REGION Network 172: M875- / M23-SWITCH ON SPINDLE FRAME BLOWING
   RUNG wire#powerrail
      Contact( "DB339_EXTENDED_M_SPARE".M_code[875] )
      wire#w1
      I_Contact( "DB371_M_UNIT_SPARE".M_CODES_SPARE.Ack_M875 )
      I_Contact( "DB2120_MPP_ITC_IPC".RESET_FAULTS )
      I_Contact( "DB371_M_UNIT_SPARE".M_CODES_SPARE.M_RESET_PULSE )
      Coil( "DB371_M_UNIT_SPARE".M_CODES_SPARE.M875 )
   END_RUNG
   RUNG wire#powerrail
      Contact( "DB371_M_UNIT_SPARE".M_CODES_SPARE.M875 )
   END_RUNG wire#w1
   // the same network as SCL:
   "DB371_M_UNIT_SPARE".M_CODES_SPARE.M875 := ("DB339_EXTENDED_M_SPARE".M_code[875] OR "DB371_M_UNIT_SPARE".M_CODES_SPARE.M875) AND NOT "DB371_M_UNIT_SPARE".M_CODES_SPARE.Ack_M875 AND NOT "DB2120_MPP_ITC_IPC".RESET_FAULTS AND NOT "DB371_M_UNIT_SPARE".M_CODES_SPARE.M_RESET_PULSE;
END_REGION

REGION Network 173: ACKNOWLEDGE M888- / ACKNOWLEDGE M23-SWITCH ON SPINDLE FRAME BLOWING
   RUNG wire#powerrail
      Contact( "M_ZERO" )
      Coil( "DB371_M_UNIT_SPARE".M_CODES_SPARE.Ack_M888 )
   END_RUNG
   // the same network as SCL:
   "DB371_M_UNIT_SPARE".M_CODES_SPARE.Ack_M888 := "M_ZERO";
END_REGION

REGION Network 174: M888- / M23-SWITCH ON SPINDLE FRAME BLOWING
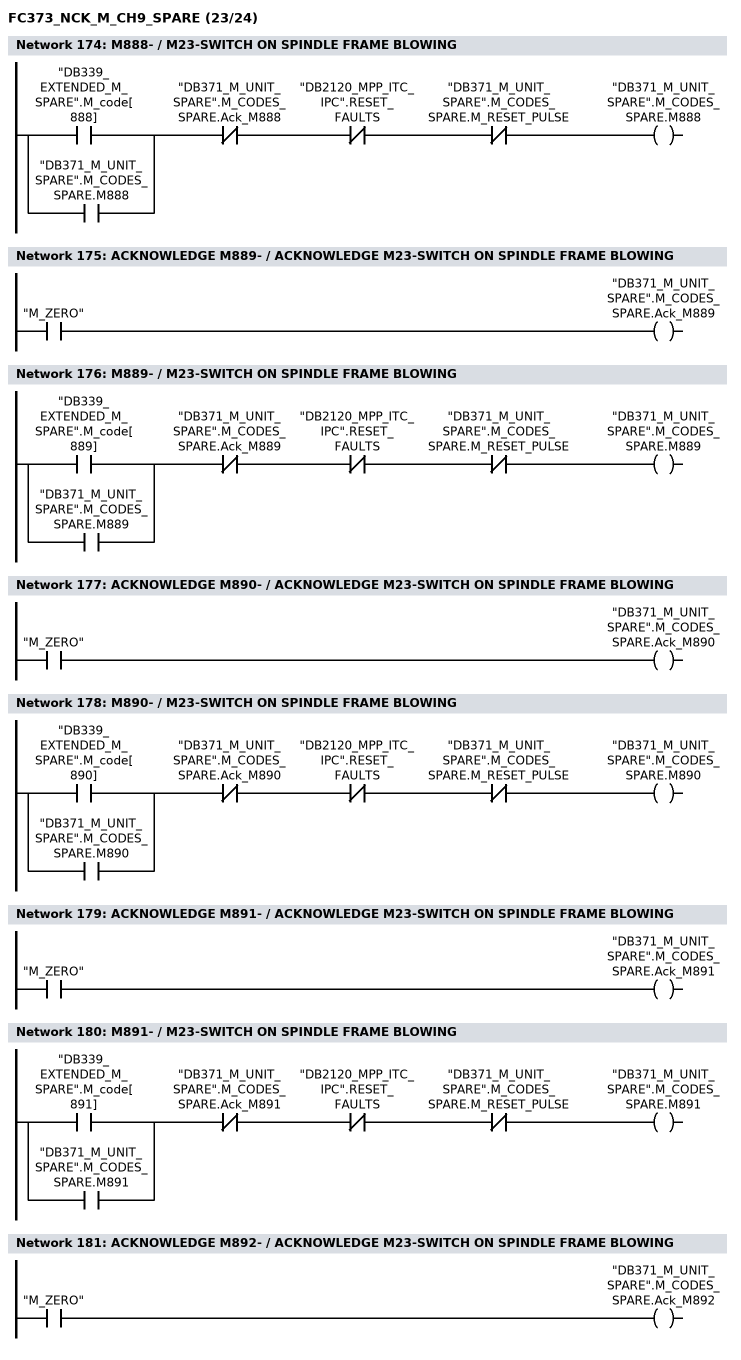
   RUNG wire#powerrail
      Contact( "DB339_EXTENDED_M_SPARE".M_code[888] )
      wire#w1
      I_Contact( "DB371_M_UNIT_SPARE".M_CODES_SPARE.Ack_M888 )
      I_Contact( "DB2120_MPP_ITC_IPC".RESET_FAULTS )
      I_Contact( "DB371_M_UNIT_SPARE".M_CODES_SPARE.M_RESET_PULSE )
      Coil( "DB371_M_UNIT_SPARE".M_CODES_SPARE.M888 )
   END_RUNG
   RUNG wire#powerrail
      Contact( "DB371_M_UNIT_SPARE".M_CODES_SPARE.M888 )
   END_RUNG wire#w1
   // the same network as SCL:
   "DB371_M_UNIT_SPARE".M_CODES_SPARE.M888 := ("DB339_EXTENDED_M_SPARE".M_code[888] OR "DB371_M_UNIT_SPARE".M_CODES_SPARE.M888) AND NOT "DB371_M_UNIT_SPARE".M_CODES_SPARE.Ack_M888 AND NOT "DB2120_MPP_ITC_IPC".RESET_FAULTS AND NOT "DB371_M_UNIT_SPARE".M_CODES_SPARE.M_RESET_PULSE;
END_REGION

REGION Network 175: ACKNOWLEDGE M889- / ACKNOWLEDGE M23-SWITCH ON SPINDLE FRAME BLOWING
   RUNG wire#powerrail
      Contact( "M_ZERO" )
      Coil( "DB371_M_UNIT_SPARE".M_CODES_SPARE.Ack_M889 )
   END_RUNG
   // the same network as SCL:
   "DB371_M_UNIT_SPARE".M_CODES_SPARE.Ack_M889 := "M_ZERO";
END_REGION

REGION Network 176: M889- / M23-SWITCH ON SPINDLE FRAME BLOWING
   RUNG wire#powerrail
      Contact( "DB339_EXTENDED_M_SPARE".M_code[889] )
      wire#w1
      I_Contact( "DB371_M_UNIT_SPARE".M_CODES_SPARE.Ack_M889 )
      I_Contact( "DB2120_MPP_ITC_IPC".RESET_FAULTS )
      I_Contact( "DB371_M_UNIT_SPARE".M_CODES_SPARE.M_RESET_PULSE )
      Coil( "DB371_M_UNIT_SPARE".M_CODES_SPARE.M889 )
   END_RUNG
   RUNG wire#powerrail
      Contact( "DB371_M_UNIT_SPARE".M_CODES_SPARE.M889 )
   END_RUNG wire#w1
   // the same network as SCL:
   "DB371_M_UNIT_SPARE".M_CODES_SPARE.M889 := ("DB339_EXTENDED_M_SPARE".M_code[889] OR "DB371_M_UNIT_SPARE".M_CODES_SPARE.M889) AND NOT "DB371_M_UNIT_SPARE".M_CODES_SPARE.Ack_M889 AND NOT "DB2120_MPP_ITC_IPC".RESET_FAULTS AND NOT "DB371_M_UNIT_SPARE".M_CODES_SPARE.M_RESET_PULSE;
END_REGION

REGION Network 177: ACKNOWLEDGE M890- / ACKNOWLEDGE M23-SWITCH ON SPINDLE FRAME BLOWING
   RUNG wire#powerrail
      Contact( "M_ZERO" )
      Coil( "DB371_M_UNIT_SPARE".M_CODES_SPARE.Ack_M890 )
   END_RUNG
   // the same network as SCL:
   "DB371_M_UNIT_SPARE".M_CODES_SPARE.Ack_M890 := "M_ZERO";
END_REGION

REGION Network 178: M890- / M23-SWITCH ON SPINDLE FRAME BLOWING
   RUNG wire#powerrail
      Contact( "DB339_EXTENDED_M_SPARE".M_code[890] )
      wire#w1
      I_Contact( "DB371_M_UNIT_SPARE".M_CODES_SPARE.Ack_M890 )
      I_Contact( "DB2120_MPP_ITC_IPC".RESET_FAULTS )
      I_Contact( "DB371_M_UNIT_SPARE".M_CODES_SPARE.M_RESET_PULSE )
      Coil( "DB371_M_UNIT_SPARE".M_CODES_SPARE.M890 )
   END_RUNG
   RUNG wire#powerrail
      Contact( "DB371_M_UNIT_SPARE".M_CODES_SPARE.M890 )
   END_RUNG wire#w1
   // the same network as SCL:
   "DB371_M_UNIT_SPARE".M_CODES_SPARE.M890 := ("DB339_EXTENDED_M_SPARE".M_code[890] OR "DB371_M_UNIT_SPARE".M_CODES_SPARE.M890) AND NOT "DB371_M_UNIT_SPARE".M_CODES_SPARE.Ack_M890 AND NOT "DB2120_MPP_ITC_IPC".RESET_FAULTS AND NOT "DB371_M_UNIT_SPARE".M_CODES_SPARE.M_RESET_PULSE;
END_REGION

REGION Network 179: ACKNOWLEDGE M891- / ACKNOWLEDGE M23-SWITCH ON SPINDLE FRAME BLOWING
   RUNG wire#powerrail
      Contact( "M_ZERO" )
      Coil( "DB371_M_UNIT_SPARE".M_CODES_SPARE.Ack_M891 )
   END_RUNG
   // the same network as SCL:
   "DB371_M_UNIT_SPARE".M_CODES_SPARE.Ack_M891 := "M_ZERO";
END_REGION

REGION Network 180: M891- / M23-SWITCH ON SPINDLE FRAME BLOWING
   RUNG wire#powerrail
      Contact( "DB339_EXTENDED_M_SPARE".M_code[891] )
      wire#w1
      I_Contact( "DB371_M_UNIT_SPARE".M_CODES_SPARE.Ack_M891 )
      I_Contact( "DB2120_MPP_ITC_IPC".RESET_FAULTS )
      I_Contact( "DB371_M_UNIT_SPARE".M_CODES_SPARE.M_RESET_PULSE )
      Coil( "DB371_M_UNIT_SPARE".M_CODES_SPARE.M891 )
   END_RUNG
   RUNG wire#powerrail
      Contact( "DB371_M_UNIT_SPARE".M_CODES_SPARE.M891 )
   END_RUNG wire#w1
   // the same network as SCL:
   "DB371_M_UNIT_SPARE".M_CODES_SPARE.M891 := ("DB339_EXTENDED_M_SPARE".M_code[891] OR "DB371_M_UNIT_SPARE".M_CODES_SPARE.M891) AND NOT "DB371_M_UNIT_SPARE".M_CODES_SPARE.Ack_M891 AND NOT "DB2120_MPP_ITC_IPC".RESET_FAULTS AND NOT "DB371_M_UNIT_SPARE".M_CODES_SPARE.M_RESET_PULSE;
END_REGION

REGION Network 181: ACKNOWLEDGE M892- / ACKNOWLEDGE M23-SWITCH ON SPINDLE FRAME BLOWING
   RUNG wire#powerrail
      Contact( "M_ZERO" )
      Coil( "DB371_M_UNIT_SPARE".M_CODES_SPARE.Ack_M892 )
   END_RUNG
   // the same network as SCL:
   "DB371_M_UNIT_SPARE".M_CODES_SPARE.Ack_M892 := "M_ZERO";
END_REGION

REGION Network 182: M892- / M23-SWITCH ON SPINDLE FRAME BLOWING
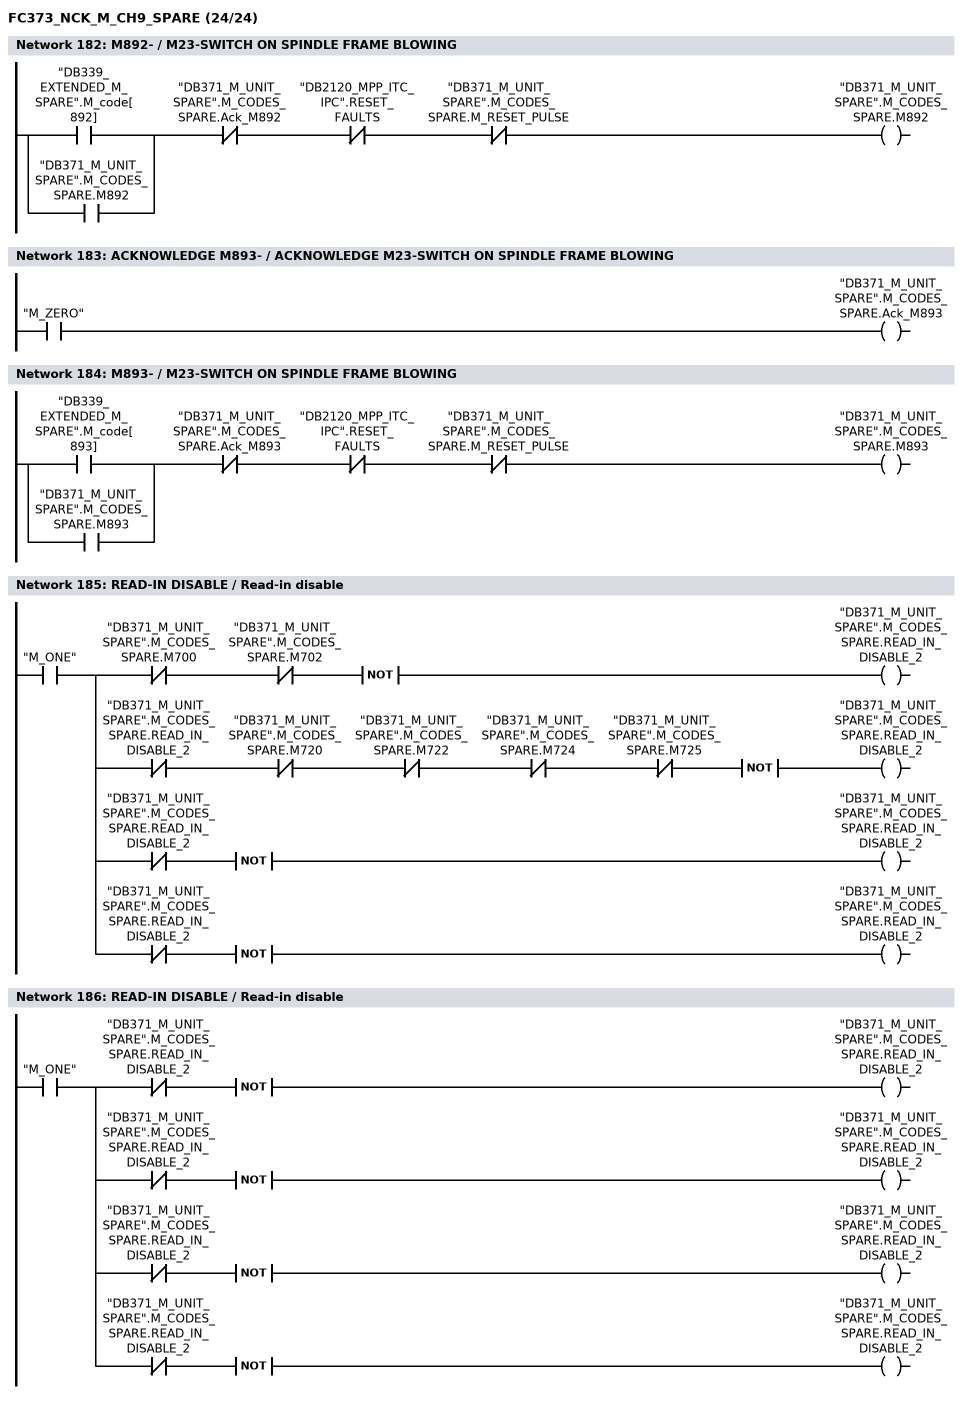
   RUNG wire#powerrail
      Contact( "DB339_EXTENDED_M_SPARE".M_code[892] )
      wire#w1
      I_Contact( "DB371_M_UNIT_SPARE".M_CODES_SPARE.Ack_M892 )
      I_Contact( "DB2120_MPP_ITC_IPC".RESET_FAULTS )
      I_Contact( "DB371_M_UNIT_SPARE".M_CODES_SPARE.M_RESET_PULSE )
      Coil( "DB371_M_UNIT_SPARE".M_CODES_SPARE.M892 )
   END_RUNG
   RUNG wire#powerrail
      Contact( "DB371_M_UNIT_SPARE".M_CODES_SPARE.M892 )
   END_RUNG wire#w1
   // the same network as SCL:
   "DB371_M_UNIT_SPARE".M_CODES_SPARE.M892 := ("DB339_EXTENDED_M_SPARE".M_code[892] OR "DB371_M_UNIT_SPARE".M_CODES_SPARE.M892) AND NOT "DB371_M_UNIT_SPARE".M_CODES_SPARE.Ack_M892 AND NOT "DB2120_MPP_ITC_IPC".RESET_FAULTS AND NOT "DB371_M_UNIT_SPARE".M_CODES_SPARE.M_RESET_PULSE;
END_REGION

REGION Network 183: ACKNOWLEDGE M893- / ACKNOWLEDGE M23-SWITCH ON SPINDLE FRAME BLOWING
   RUNG wire#powerrail
      Contact( "M_ZERO" )
      Coil( "DB371_M_UNIT_SPARE".M_CODES_SPARE.Ack_M893 )
   END_RUNG
   // the same network as SCL:
   "DB371_M_UNIT_SPARE".M_CODES_SPARE.Ack_M893 := "M_ZERO";
END_REGION

REGION Network 184: M893- / M23-SWITCH ON SPINDLE FRAME BLOWING
   RUNG wire#powerrail
      Contact( "DB339_EXTENDED_M_SPARE".M_code[893] )
      wire#w1
      I_Contact( "DB371_M_UNIT_SPARE".M_CODES_SPARE.Ack_M893 )
      I_Contact( "DB2120_MPP_ITC_IPC".RESET_FAULTS )
      I_Contact( "DB371_M_UNIT_SPARE".M_CODES_SPARE.M_RESET_PULSE )
      Coil( "DB371_M_UNIT_SPARE".M_CODES_SPARE.M893 )
   END_RUNG
   RUNG wire#powerrail
      Contact( "DB371_M_UNIT_SPARE".M_CODES_SPARE.M893 )
   END_RUNG wire#w1
   // the same network as SCL:
   "DB371_M_UNIT_SPARE".M_CODES_SPARE.M893 := ("DB339_EXTENDED_M_SPARE".M_code[893] OR "DB371_M_UNIT_SPARE".M_CODES_SPARE.M893) AND NOT "DB371_M_UNIT_SPARE".M_CODES_SPARE.Ack_M893 AND NOT "DB2120_MPP_ITC_IPC".RESET_FAULTS AND NOT "DB371_M_UNIT_SPARE".M_CODES_SPARE.M_RESET_PULSE;
END_REGION

REGION Network 185: READ-IN DISABLE / Read-in disable
   RUNG wire#powerrail
      Contact( "M_ONE" )
      wire#w1
      I_Contact( "DB371_M_UNIT_SPARE".M_CODES_SPARE.M700 )
      I_Contact( "DB371_M_UNIT_SPARE".M_CODES_SPARE.M702 )
      Not()
      Coil( "DB371_M_UNIT_SPARE".M_CODES_SPARE.READ_IN_DISABLE_2 )
   END_RUNG
   RUNG wire#w1
      I_Contact( "DB371_M_UNIT_SPARE".M_CODES_SPARE.READ_IN_DISABLE_2 )
      I_Contact( "DB371_M_UNIT_SPARE".M_CODES_SPARE.M720 )
      I_Contact( "DB371_M_UNIT_SPARE".M_CODES_SPARE.M722 )
      I_Contact( "DB371_M_UNIT_SPARE".M_CODES_SPARE.M724 )
      I_Contact( "DB371_M_UNIT_SPARE".M_CODES_SPARE.M725 )
      Not()
      Coil( "DB371_M_UNIT_SPARE".M_CODES_SPARE.READ_IN_DISABLE_2 )
   END_RUNG
   RUNG wire#w1
      I_Contact( "DB371_M_UNIT_SPARE".M_CODES_SPARE.READ_IN_DISABLE_2 )
      Not()
      Coil( "DB371_M_UNIT_SPARE".M_CODES_SPARE.READ_IN_DISABLE_2 )
   END_RUNG
   RUNG wire#w1
      I_Contact( "DB371_M_UNIT_SPARE".M_CODES_SPARE.READ_IN_DISABLE_2 )
      Not()
      Coil( "DB371_M_UNIT_SPARE".M_CODES_SPARE.READ_IN_DISABLE_2 )
   END_RUNG
   // the same network as SCL:
   "DB371_M_UNIT_SPARE".M_CODES_SPARE.READ_IN_DISABLE_2 := NOT ("M_ONE" AND NOT "DB371_M_UNIT_SPARE".M_CODES_SPARE.M700 AND NOT "DB371_M_UNIT_SPARE".M_CODES_SPARE.M702);
   "DB371_M_UNIT_SPARE".M_CODES_SPARE.READ_IN_DISABLE_2 := NOT ("M_ONE" AND NOT "DB371_M_UNIT_SPARE".M_CODES_SPARE.READ_IN_DISABLE_2 AND NOT "DB371_M_UNIT_SPARE".M_CODES_SPARE.M720 AND NOT "DB371_M_UNIT_SPARE".M_CODES_SPARE.M722 AND NOT "DB371_M_UNIT_SPARE".M_CODES_SPARE.M724 AND NOT "DB371_M_UNIT_SPARE".M_CODES_SPARE.M725);
   "DB371_M_UNIT_SPARE".M_CODES_SPARE.READ_IN_DISABLE_2 := NOT ("M_ONE" AND NOT "DB371_M_UNIT_SPARE".M_CODES_SPARE.READ_IN_DISABLE_2);
   "DB371_M_UNIT_SPARE".M_CODES_SPARE.READ_IN_DISABLE_2 := NOT ("M_ONE" AND NOT "DB371_M_UNIT_SPARE".M_CODES_SPARE.READ_IN_DISABLE_2);
END_REGION

REGION Network 186: READ-IN DISABLE / Read-in disable
   RUNG wire#powerrail
      Contact( "M_ONE" )
      wire#w1
      I_Contact( "DB371_M_UNIT_SPARE".M_CODES_SPARE.READ_IN_DISABLE_2 )
      Not()
      Coil( "DB371_M_UNIT_SPARE".M_CODES_SPARE.READ_IN_DISABLE_2 )
   END_RUNG
   RUNG wire#w1
      I_Contact( "DB371_M_UNIT_SPARE".M_CODES_SPARE.READ_IN_DISABLE_2 )
      Not()
      Coil( "DB371_M_UNIT_SPARE".M_CODES_SPARE.READ_IN_DISABLE_2 )
   END_RUNG
   RUNG wire#w1
      I_Contact( "DB371_M_UNIT_SPARE".M_CODES_SPARE.READ_IN_DISABLE_2 )
      Not()
      Coil( "DB371_M_UNIT_SPARE".M_CODES_SPARE.READ_IN_DISABLE_2 )
   END_RUNG
   RUNG wire#w1
      I_Contact( "DB371_M_UNIT_SPARE".M_CODES_SPARE.READ_IN_DISABLE_2 )
      Not()
      Coil( "DB371_M_UNIT_SPARE".M_CODES_SPARE.READ_IN_DISABLE_2 )
   END_RUNG
   // the same network as SCL:
   "DB371_M_UNIT_SPARE".M_CODES_SPARE.READ_IN_DISABLE_2 := NOT ("M_ONE" AND NOT "DB371_M_UNIT_SPARE".M_CODES_SPARE.READ_IN_DISABLE_2);
   "DB371_M_UNIT_SPARE".M_CODES_SPARE.READ_IN_DISABLE_2 := NOT ("M_ONE" AND NOT "DB371_M_UNIT_SPARE".M_CODES_SPARE.READ_IN_DISABLE_2);
   "DB371_M_UNIT_SPARE".M_CODES_SPARE.READ_IN_DISABLE_2 := NOT ("M_ONE" AND NOT "DB371_M_UNIT_SPARE".M_CODES_SPARE.READ_IN_DISABLE_2);
   "DB371_M_UNIT_SPARE".M_CODES_SPARE.READ_IN_DISABLE_2 := NOT ("M_ONE" AND NOT "DB371_M_UNIT_SPARE".M_CODES_SPARE.READ_IN_DISABLE_2);
END_REGION
END_FUNCTION
